INTERFACE IProcess EXTENDS IStation

PROPERTY EndPosition : MC_LREAL
GET
END_GET
SET
END_SET
END_PROPERTY

PROPERTY IsProcess : booL
GET
END_GET
SET
END_SET
END_PROPERTY

PROPERTY ProcessVelocity : mc_lreal
GET
END_GET
SET
END_SET
END_PROPERTY

PROPERTY StartPosition : MC_LREAL
GET
END_GET
SET
END_SET
END_PROPERTY

END_INTERFACE

(* stored: Version 1.1.0.1, ProductVersion 3.1.4024.12
   Itf IProcess: Id {35f38492-ddb4-43cb-90ed-57490b1c2a0f}
   Property EndPosition: Id {dd6f2210-a4af-4fbc-a10a-6e02b45480ee}
   Get Get: Id {31f9cf28-dd57-4d20-ace6-7cac7fc9bf57}
   Set Set: Id {b3f53b23-605e-4691-b489-df326d97e83e}
   Property IsProcess: Id {715b1fa2-b476-4fb4-a0e0-f20bf4d903ee}
   Get Get: Id {755e0674-f78a-4a37-8b52-990c4b63efad}
   Set Set: Id {c6802322-6194-46c4-a3cb-ca06cc0cd717}
   Property ProcessVelocity: Id {4148105b-d9b1-443c-b3c0-196030eb7c2f}
   Get Get: Id {4f40390c-f906-437a-882e-04f737dbad29}
   Set Set: Id {f38d7b69-5b1f-4bd3-9e08-ad34bc533051}
   Property StartPosition: Id {98da2cda-f61a-4ce0-b8d5-531a68fd5332}
   Get Get: Id {fcc845e3-1036-4df4-a77e-62ba44d37e6e}
   Set Set: Id {b37b04b9-b5ec-4bb3-8455-6bb9205981a2} *)
